ABB RobotStudio station: Celda_4_Enero.rsstn

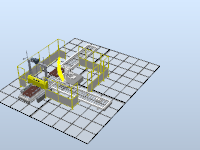
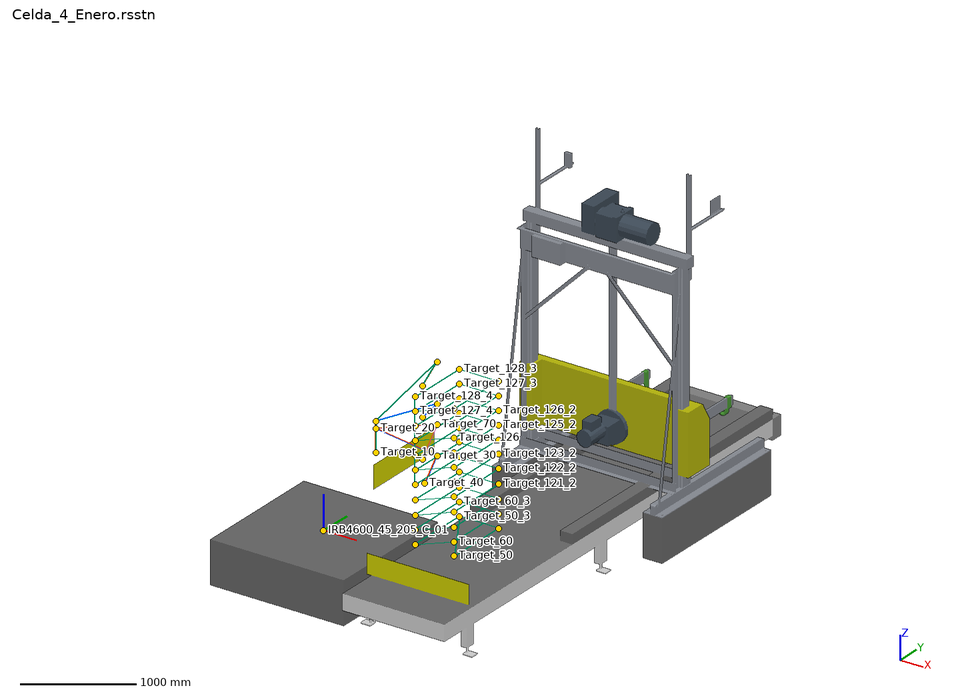
[picture v1: parts stored in the station drawn from their meshes, with robot base, taught points and paths (robot models come from the ABB library and are not in the file)]
Station Celda (saved by RobotStudio 21.3.9648.0)
Controller Controlador1, task T_ROB1: task frame (RAPID world) sits at (0, 0, 435) mm in the station
Controller Controlador1
  mechanical unit ROB_1: IRB4600_45_205_C_01, 6 joints, base frame (0, 0, 0) mm
Layout (positions relative to the parent item):
  - Entrada de canastillas [smart component]
      signals: DO Canasta_ok, DI Soltar, DI Agarrar, DO Agarrado, DI Pallet_fisica
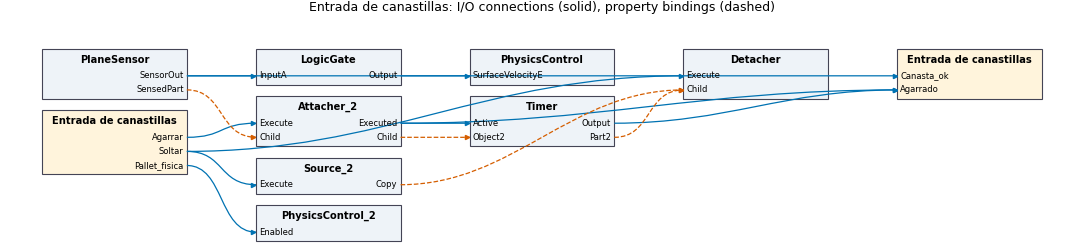
      connections:
        PlaneSensor.SensorOut -> LogicGate.InputA
        LogicGate.Output -> PhysicsControl.SurfaceVelocityEnabled
        PlaneSensor.SensorOut -> Entrada de canastillas.Canasta_ok
        Entrada de canastillas.Agarrar -> Attacher_2.Execute
        Attacher_2.Executed -> Timer.Active
        Timer.Output -> Entrada de canastillas.Agarrado
        Attacher_2.Executed -> Entrada de canastillas.Agarrado
        Entrada de canastillas.Soltar -> Detacher.Execute
        Entrada de canastillas.Pallet_fisica -> PhysicsControl_2.Enabled
        Entrada de canastillas.Soltar -> Source_2.Execute
        PlaneSensor.SensedPart => Attacher_2.Child
        CollisionSensor.Part2 => Detacher.Child
        Attacher_2.Child => CollisionSensor.Object2
        Source_2.Copy => Detacher.Child
    - Source_2 [smart component, from Components\Source.rslib]
        properties: Source=Plastic crate; Copy=(none); Parent=(none); Position=[-2.8 1.3 0.565]; Orientation=[3.14159265358979 0 0]; Transient=false; PhysicsBehavior=3
    - PlaneSensor [smart component, from Components\PlaneSensor.rslib]
        properties: Origin=[-0.076705 1.76 0.467165]; Axis1=[0 -0.91 0]; Axis2=[-5E-06 0 0.232835]; SensedPart=(none)
      - _sensorPart_ [part], size 0 x 910 x 232.8 mm
    - PhysicsControl [smart component, from Components\PhysicsControl.rslib]
        properties: Object=Banda_Canastas; Behavior=2; SurfaceVelocity=0.7
    - LogicGate [smart component, from Components\LogicGate.rslib]
        properties: Operator=NOT; Delay=0
    - Attacher_2 [smart component, from Components\Attacher.rslib]
        properties: Parent=MyNewTool; Flange=0; Child=(none); Mount=false; Offset=[0 0 0]; Orientation=[0 0 0]
    - Detacher [smart component, from Components\Detacher.rslib]
        properties: Child=(none); KeepPosition=true
    - PhysicsControl_2 [smart component, from Components\PhysicsControl.rslib]
        properties: Object=Euro Pallet; Behavior=3; SurfaceVelocity=0
  - IRB4600_45_205_C_01 [mechanism, from Robots\IRB4600_45_205_C_G_01.rslib] at (0, 0, 435) mm; joint values [1.8433, 0.6847, 0.3992, 0, 0.4869, -1.2983] (rad or m)
  - MyNewTool [mechanism] at (-362.82, 1298.26, 725.56) mm, rotated rx -180 ry 0 rz 0 deg
      TCP Gripper at (0, 0, 166) mm
      links: NewGripper
  - Perimetro [graphiccomponentgroup]
    - Fence_2503 [graphiccomponentgroup, from Equipment\Fence_2500.rslib] at (3000, 238.8, 0) mm
      - Body 1 [part, from Equipment\Fence_2500.rslib]
      - Body 2 [part, from Equipment\Fence_2500.rslib]
    - Fence_2502 [graphiccomponentgroup, from Equipment\Fence_2500.rslib] at (3000, -2235.69, 0) mm
      - Body 1 [part, from Equipment\Fence_2500.rslib]
      - Body 2 [part, from Equipment\Fence_2500.rslib]
    - Fence_2500 [graphiccomponentgroup, from Equipment\Fence_2500.rslib] at (-2079.28, 2740, 0) mm, rotated rx 0 ry 0 rz -90 deg
      - Body 1 [part, from Equipment\Fence_2500.rslib]
      - Body 2 [part, from Equipment\Fence_2500.rslib]
    - Fence_740_12 [graphiccomponentgroup, from Equipment\Fence_740.rslib] at (3000, -2297.98, 0) mm, rotated rx 0 ry 0 rz 90 deg
      - Body 1 [part, from Equipment\Fence_740.rslib]
      - Body 2 [part, from Equipment\Fence_740.rslib]
    - Fence_740_11 [graphiccomponentgroup, from Equipment\Fence_740.rslib] at (-2100, -2267.47, 0) mm
      - Body 1 [part, from Equipment\Fence_740.rslib]
      - Body 2 [part, from Equipment\Fence_740.rslib]
    - Fence_740_10 [graphiccomponentgroup, from Equipment\Fence_740.rslib] at (82.68, -2200, 0) mm, rotated rx 0 ry 0 rz -90 deg
      - Body 1 [part, from Equipment\Fence_740.rslib]
      - Body 2 [part, from Equipment\Fence_740.rslib]
    - Fence_740_9 [graphiccomponentgroup, from Equipment\Fence_740.rslib] at (-657.15, -2200, 0) mm, rotated rx 0 ry 0 rz -90 deg
      - Body 1 [part, from Equipment\Fence_740.rslib]
      - Body 2 [part, from Equipment\Fence_740.rslib]
    - Fence_740_8 [graphiccomponentgroup, from Equipment\Fence_740.rslib] at (-1386.41, -2200, 0) mm, rotated rx 0 ry 0 rz -90 deg
      - Body 1 [part, from Equipment\Fence_740.rslib]
      - Body 2 [part, from Equipment\Fence_740.rslib]
    - Fence_740_4 [graphiccomponentgroup, from Equipment\Fence_740.rslib] at (-2153.49, -2200, 0) mm, rotated rx 0 ry 0 rz -90 deg
      - Body 1 [part, from Equipment\Fence_740.rslib]
      - Body 2 [part, from Equipment\Fence_740.rslib]
    - Fence_740_3 [graphiccomponentgroup, from Equipment\Fence_740.rslib] at (-2100, -1490.03, 0) mm
      - Body 1 [part, from Equipment\Fence_740.rslib]
      - Body 2 [part, from Equipment\Fence_740.rslib]
    - Fence_740_2 [graphiccomponentgroup, from Equipment\Fence_740.rslib] at (3000, 2740, 0) mm, rotated rx 0 ry 0 rz 90 deg
      - Body 1 [part, from Equipment\Fence_740.rslib]
      - Body 2 [part, from Equipment\Fence_740.rslib]
    - Fence_740 [graphiccomponentgroup, from Equipment\Fence_740.rslib] at (-2100, 2000, 0) mm
      - Body 1 [part, from Equipment\Fence_740.rslib]
      - Body 2 [part, from Equipment\Fence_740.rslib]
    - Gate [graphiccomponentgroup, from Equipment\Fence_Gate.rslib] at (-2100, 728.56, 0) mm, rotated rx 0 ry 0 rz 180 deg
      - Body 1 [part, from Equipment\Fence_Gate.rslib]
      - Body 2 [part, from Equipment\Fence_Gate.rslib]
      - Body 3 [part, from Equipment\Fence_Gate.rslib]
    - Part_2 [part] at (-700, -700, 0) mm, size 1400 x 1400 x 435 mm
    - Soporte1 [part], size 200 x 1630 x 430 mm
    - Soporte2 [part], size 200 x 1630 x 430 mm
  - Plastic crate [part] at (-3299.78, 1300.28, 558.99) mm, rotated rx 179.83 ry 0.16 rz 0.13 deg, size 603.9 x 403.9 x 145.1 mm
  - Entrada de pallets [smart component]
      connections:
        PlaneSensor.SensorOut -> Source.Execute
        PlaneSensor.SensorOut -> LogicGate.InputA
        LogicGate.Output -> PhysicsControl.SurfaceVelocityEnabled
    - Source [smart component, from Components\Source.rslib]
        properties: Source=Euro Pallet; Copy=Euro Pallet_84; Parent=(none); Position=[1.75 2.6 0.44]; Orientation=[0 0 1.5707963267949]; Transient=false; PhysicsBehavior=3
    - PlaneSensor [smart component, from Components\PlaneSensor.rslib]
        properties: Origin=[0.84 -0.55 0.475]; Axis1=[1.07 0 0]; Axis2=[0 0 0.2]; SensedPart=Body 1
      - _sensorPart_ [part], size 1070 x 0 x 200 mm
    - PhysicsControl [smart component, from Components\PhysicsControl.rslib]
        properties: Object=Banda_P_Entrada_S; Behavior=1; SurfaceVelocity=0.5
    - LogicGate [smart component, from Components\LogicGate.rslib]
        properties: Operator=NOT; Delay=0
  - Bandas [graphiccomponentgroup]
    - Banda_Canastas [part, from Equipment\Conveyor 950 4800 h2.rslib] at (-4200, 850, 0) mm
    - Banda_P_Entrada [part] at (900, 4000, 0) mm, rotated rx 0 ry 0 rz -90 deg, size 5049.9 x 1178.5 x 441.9 mm
    - Banda_P_Entrada_S [part], size 1070 x 4920 x 1 mm
    - Banda_P_Salida [part, from Equipment\Conveyor 950 4000 h2.rslib] at (900, -1050, 0) mm, rotated rx 0 ry 0 rz -90 deg
    - Barrera1 [part], size 130 x 3000 x 100 mm
    - Barrera2 [part] at (-2, 0, 0) mm, size 123 x 3000 x 100 mm
  - Euro Pallet [graphiccomponentgroup, from Equipment\Euro Pallet.rslib] at (1762.72, -569.55, 439.14) mm, rotated rx 0 ry 0 rz 89.52 deg
    - Body 1 [part, from Equipment\Euro Pallet.rslib]
  - Euro Pallet_2 [graphiccomponentgroup, from Equipment\Euro Pallet.rslib] at (1757, -550, 440) mm, rotated rx 0 ry 0 rz 90 deg
    - Body 1 [part, from Equipment\Euro Pallet.rslib]
  - DispenserPallet [part] at (1350, 3500, 430) mm, rotated rx 90 ry 0 rz 180 deg, size 1784 x 3045 x 1697.6 mm
  - Euro Pallet_84 [graphiccomponentgroup, from Equipment\Euro Pallet.rslib] at (1773.49, 2601.34, 439.14) mm, rotated rx 0 ry 0 rz 90.55 deg
    - Body 1 [part, from Equipment\Euro Pallet.rslib]
Attachment: MyNewTool is attached to IRB4600_45_205_C_01 / Link6
Attachment: PhysicsControl is attached to Banda_Canastas
Station signals: DO Canasta_ok
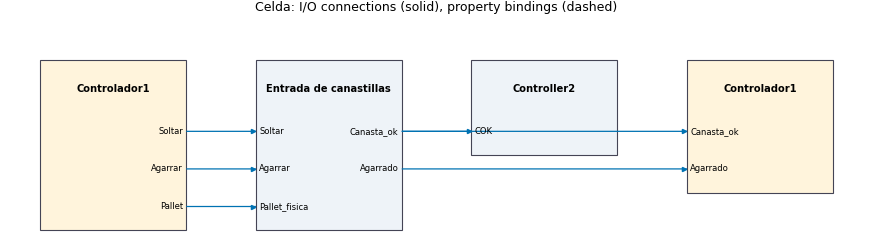
Station logic (signal -> signal, property => property):
  Entrada de canastillas.Canasta_ok -> Controller2.COK
  Entrada de canastillas.Canasta_ok -> Controlador1.Canasta_ok
  Controlador1.Soltar -> Entrada de canastillas.Soltar
  Controlador1.Agarrar -> Entrada de canastillas.Agarrar
  Entrada de canastillas.Agarrado -> Controlador1.Agarrado
  Controlador1.Pallet -> Entrada de canastillas.Pallet_fisica
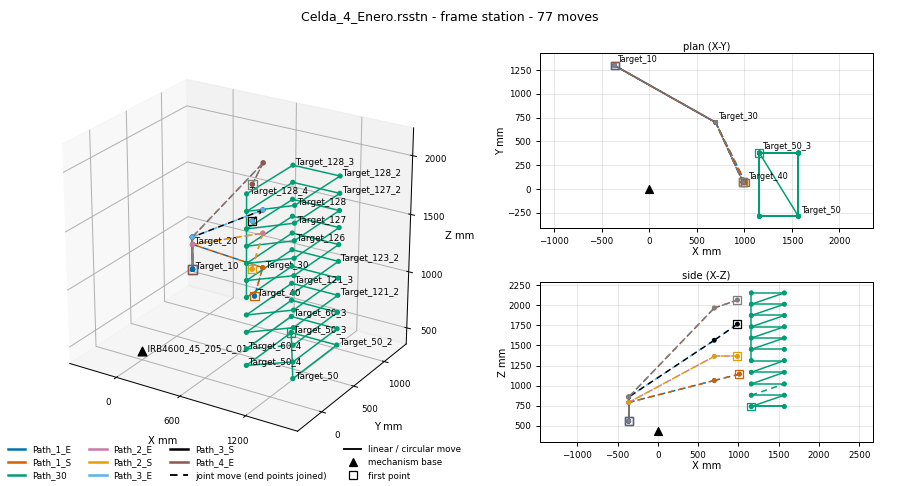
[picture p0: tool path of Celda_4_Enero.rsstn in frame station, 77 of 77 moves have a stored position in this frame; points joined in program order, loops and branches not executed]
Targets, tools, work objects and paths stored in the station, written as RAPID:
! task (no controller)
MODULE CalibData
  TASK PERS wobjdata Workobject_1:=[FALSE,TRUE,"",[[0,0,0],[1,0,0,0]],[[0,0,0],[1,0,0,0]]];
ENDMODULE

! task T_ROB1
MODULE CalibData
  PERS tooldata Gripper:=[TRUE,[[0,0,166],[1,0,0,0]],[27.5,[0,0,86.1],[1,0,0,0],0.589498,1.412,1.775]];
  TASK PERS wobjdata Workobject_1:=[FALSE,TRUE,"",[[0,0,0],[1,0,0,0]],[[0,0,0],[1,0,0,0]]];
ENDMODULE

! task T_ROB1
MODULE Module1
  CONST robtarget Target_10:=[[-362.824,1298.255,124.558],[0,1,0,0],[0,0,0,0],[9E+09,9E+09,9E+09,9E+09,9E+09,9E+09]];
  CONST robtarget Target_30:=[[699.999971128,699.99999496,629.43677315],[0.000000013,0.714564003,0.699570072,0.000000004],[0,-1,-2,0],[9E+09,9E+09,9E+09,9E+09,9E+09,9E+09]];
  CONST robtarget Target_50:=[[1570,-287,307],[0,0.707106781,0.707106781,0],[-1,0,0,0],[9E+09,9E+09,9E+09,9E+09,9E+09,9E+09]];
  CONST robtarget Target_60:=[[1570,-287,447],[0,0.707106781,0.707106781,0],[0,0,0,0],[9E+09,9E+09,9E+09,9E+09,9E+09,9E+09]];
  CONST robtarget Target_50_3:=[[1160,378,307],[0,0.707106781,0.707106781,0],[0,0,0,0],[9E+09,9E+09,9E+09,9E+09,9E+09,9E+09]];
  CONST robtarget Target_50_4:=[[1160,-287,307],[0,0.707106781,0.707106781,0],[-1,0,0,0],[9E+09,9E+09,9E+09,9E+09,9E+09,9E+09]];
  CONST robtarget Target_50_2:=[[1570,378,307],[0,0.707106781,0.707106781,0],[0,0,0,0],[9E+09,9E+09,9E+09,9E+09,9E+09,9E+09]];
  CONST robtarget Target_10_2:=[[-362.824,1298.255,424.558],[-0.000000012,0.998529603,-0.054209154,0.000000007],[1,0,-1,0],[9E+09,9E+09,9E+09,9E+09,9E+09,9E+09]];
  CONST robtarget Target_60_2:=[[1570,378,447],[0,0.707106781,0.707106781,0],[0,0,1,0],[9E+09,9E+09,9E+09,9E+09,9E+09,9E+09]];
  CONST robtarget Target_60_3:=[[1160,378,447],[0,0.707106781,0.707106781,0],[0,0,1,0],[9E+09,9E+09,9E+09,9E+09,9E+09,9E+09]];
  CONST robtarget Target_60_4:=[[1160,-287,447],[0,0.707106781,0.707106781,0],[-1,0,0,0],[9E+09,9E+09,9E+09,9E+09,9E+09,9E+09]];
  CONST robtarget Target_120_2:=[[1570,378,587],[0,0.707106781,0.707106781,0],[0,0,1,0],[9E+09,9E+09,9E+09,9E+09,9E+09,9E+09]];
  CONST robtarget Target_120_3:=[[1160,378,587],[0,0.707106781,0.707106781,0],[0,0,1,0],[9E+09,9E+09,9E+09,9E+09,9E+09,9E+09]];
  CONST robtarget Target_120_4:=[[1160,-287,587],[0,0.707106781,0.707106781,0],[-1,0,0,0],[9E+09,9E+09,9E+09,9E+09,9E+09,9E+09]];
  CONST robtarget Target_121:=[[1570,-287,732],[0,0.707106781,0.707106781,0],[-1,0,0,0],[9E+09,9E+09,9E+09,9E+09,9E+09,9E+09]];
  CONST robtarget Target_121_2:=[[1570,378,732],[0,0.707106781,0.707106781,0],[0,0,1,0],[9E+09,9E+09,9E+09,9E+09,9E+09,9E+09]];
  CONST robtarget Target_121_3:=[[1160,378,732],[0,0.707106781,0.707106781,0],[0,0,1,0],[9E+09,9E+09,9E+09,9E+09,9E+09,9E+09]];
  CONST robtarget Target_121_4:=[[1160,-287,732],[0,0.707106781,0.707106781,0],[-1,0,0,0],[9E+09,9E+09,9E+09,9E+09,9E+09,9E+09]];
  CONST robtarget Target_122:=[[1570,-287,877],[0,0.707106781,0.707106781,0],[-1,0,0,0],[9E+09,9E+09,9E+09,9E+09,9E+09,9E+09]];
  CONST robtarget Target_122_2:=[[1570,378,877],[0,0.707106781,0.707106781,0],[0,0,1,0],[9E+09,9E+09,9E+09,9E+09,9E+09,9E+09]];
  CONST robtarget Target_122_3:=[[1160,378,877],[0,0.707106781,0.707106781,0],[0,0,1,0],[9E+09,9E+09,9E+09,9E+09,9E+09,9E+09]];
  CONST robtarget Target_122_4:=[[1160,-287,877],[0,0.707106781,0.707106781,0],[-1,0,0,0],[9E+09,9E+09,9E+09,9E+09,9E+09,9E+09]];
  CONST robtarget Target_70_2:=[[699.999994937,700.000110159,929.436793547],[-0.000000013,0.714564003,0.699570072,0.000000004],[0,-1,-2,0],[9E+09,9E+09,9E+09,9E+09,9E+09,9E+09]];
  CONST robtarget Target_123:=[[1570,-287,1017],[0,0.707106781,0.707106781,0],[-1,0,0,0],[9E+09,9E+09,9E+09,9E+09,9E+09,9E+09]];
  CONST robtarget Target_124:=[[1570,-287,1157],[0,0.707106781,0.707106781,0],[-1,0,0,0],[9E+09,9E+09,9E+09,9E+09,9E+09,9E+09]];
  CONST robtarget Target_125:=[[1570,-287,1297],[0,0.707106781,0.707106781,0],[-1,0,0,0],[9E+09,9E+09,9E+09,9E+09,9E+09,9E+09]];
  CONST robtarget Target_126:=[[1570,-287,1437],[0,0.707106781,0.707106781,0],[-1,0,0,0],[9E+09,9E+09,9E+09,9E+09,9E+09,9E+09]];
  CONST robtarget Target_127:=[[1570,-287,1577],[0,0.707106781,0.707106781,0],[-1,0,0,0],[9E+09,9E+09,9E+09,9E+09,9E+09,9E+09]];
  CONST robtarget Target_128:=[[1570,-287,1717],[0,0.707106781,0.707106781,0],[-1,0,0,0],[9E+09,9E+09,9E+09,9E+09,9E+09,9E+09]];
  CONST robtarget Target_123_2:=[[1570,378,1017],[0,0.707106781,0.707106781,0],[0,0,1,0],[9E+09,9E+09,9E+09,9E+09,9E+09,9E+09]];
  CONST robtarget Target_124_2:=[[1570,378,1157],[0,0.707106781,0.707106781,0],[0,0,1,0],[9E+09,9E+09,9E+09,9E+09,9E+09,9E+09]];
  CONST robtarget Target_125_2:=[[1570,378,1297],[0,0.707106781,0.707106781,0],[0,0,1,0],[9E+09,9E+09,9E+09,9E+09,9E+09,9E+09]];
  CONST robtarget Target_126_2:=[[1570,378,1437],[0,0.707106781,0.707106781,0],[0,0,1,0],[9E+09,9E+09,9E+09,9E+09,9E+09,9E+09]];
  CONST robtarget Target_127_2:=[[1570,378,1577],[0,0.707106781,0.707106781,0],[0,0,1,0],[9E+09,9E+09,9E+09,9E+09,9E+09,9E+09]];
  CONST robtarget Target_128_2:=[[1570,378,1717],[0,0.707106781,0.707106781,0],[0,0,1,0],[9E+09,9E+09,9E+09,9E+09,9E+09,9E+09]];
  CONST robtarget Target_123_3:=[[1160,378,1017],[0,0.707106781,0.707106781,0],[0,0,1,0],[9E+09,9E+09,9E+09,9E+09,9E+09,9E+09]];
  CONST robtarget Target_124_3:=[[1160,378,1157],[0,0.707106781,0.707106781,0],[0,0,1,0],[9E+09,9E+09,9E+09,9E+09,9E+09,9E+09]];
  CONST robtarget Target_125_3:=[[1160,378,1297],[0,0.707106781,0.707106781,0],[0,0,1,0],[9E+09,9E+09,9E+09,9E+09,9E+09,9E+09]];
  CONST robtarget Target_126_3:=[[1160,378,1437],[0,0.707106781,0.707106781,0],[0,0,1,0],[9E+09,9E+09,9E+09,9E+09,9E+09,9E+09]];
  CONST robtarget Target_127_3:=[[1160,378,1577],[0,0.707106781,0.707106781,0],[0,0,1,0],[9E+09,9E+09,9E+09,9E+09,9E+09,9E+09]];
  CONST robtarget Target_128_3:=[[1160,378,1717],[0,0.707106781,0.707106781,0],[0,0,1,0],[9E+09,9E+09,9E+09,9E+09,9E+09,9E+09]];
  CONST robtarget Target_123_4:=[[1160,-287,1017],[0,0.707106781,0.707106781,0],[-1,0,0,0],[9E+09,9E+09,9E+09,9E+09,9E+09,9E+09]];
  CONST robtarget Target_124_4:=[[1160,-287,1157],[0,0.707106781,0.707106781,0],[-1,0,0,0],[9E+09,9E+09,9E+09,9E+09,9E+09,9E+09]];
  CONST robtarget Target_125_4:=[[1160,-287,1297],[0,0.707106781,0.707106781,0],[-1,0,0,0],[9E+09,9E+09,9E+09,9E+09,9E+09,9E+09]];
  CONST robtarget Target_126_4:=[[1160,-287,1437],[0,0.707106781,0.707106781,0],[-1,0,0,0],[9E+09,9E+09,9E+09,9E+09,9E+09,9E+09]];
  CONST robtarget Target_127_4:=[[1160,-287,1577],[0,0.707106781,0.707106781,0],[-1,0,0,0],[9E+09,9E+09,9E+09,9E+09,9E+09,9E+09]];
  CONST robtarget Target_128_4:=[[1160,-287,1717],[0,0.707106781,0.707106781,0],[-1,2,-2,1],[9E+09,9E+09,9E+09,9E+09,9E+09,9E+09]];
  CONST robtarget Target_10_3:=[[-362.824,1298.255,124.558],[0,1,0,0],[0,0,0,0],[9E+09,9E+09,9E+09,9E+09,9E+09,9E+09]];
  CONST robtarget Target_20_2:=[[123.294942114,850.000075451,439.015995707],[0.000000013,0.714564003,0.699570072,0.000000004],[0,0,1,0],[9E+09,9E+09,9E+09,9E+09,9E+09,9E+09]];
  CONST robtarget Target_10_4:=[[-362.824,1298.255,124.558],[0,1,0,0],[0,0,0,0],[9E+09,9E+09,9E+09,9E+09,9E+09,9E+09]];
  CONST robtarget Target_40:=[[1012.141019914,68.859882763,709.132396194],[0.000000014,0.714564001,0.699570074,0.000000028],[0,0,-3,0],[9E+09,9E+09,9E+09,9E+09,9E+09,9E+09]];
  CONST robtarget Target_20:=[[-361.331074857,1298.255015663,357.504486712],[0.000000006,0.937903782,0.346895511,-0.000000016],[1,0,-2,0],[9E+09,9E+09,9E+09,9E+09,9E+09,9E+09]];
  CONST robtarget Target_70:=[[700.00000486,700.000107801,929.436838226],[0.000000013,0.714563971,0.699570104,-0.000000014],[0,-1,-3,0],[9E+09,9E+09,9E+09,9E+09,9E+09,9E+09]];
  CONST robtarget Target_40_2:=[[987.25590411,72.978878039,929.436817205],[0.00000003,0.714563992,0.699570083,0.000000024],[0,-1,1,0],[9E+09,9E+09,9E+09,9E+09,9E+09,9E+09]];
  CONST robtarget Target_30_2:=[[699.999992444,700.000011939,1129.436971585],[0.000000013,0.714563994,0.699570081,-0.000000007],[0,-1,-3,0],[9E+09,9E+09,9E+09,9E+09,9E+09,9E+09]];
  CONST robtarget Target_40_2_2:=[[987.255899553,72.978877702,1329.437041905],[0.00000002,0.714563994,0.699570081,0.000000013],[0,-1,1,0],[9E+09,9E+09,9E+09,9E+09,9E+09,9E+09]];
  CONST robtarget Target_30_3:=[[699.999994518,700.000014013,1529.436978926],[0.000000013,0.714563998,0.699570077,0.000000012],[0,-1,-3,0],[9E+09,9E+09,9E+09,9E+09,9E+09,9E+09]];
  CONST robtarget Target_40_2_3:=[[987.255908383,72.978882952,1629.436986878],[-0.000000004,0.714563993,0.699570082,0.000000014],[0,0,1,0],[9E+09,9E+09,9E+09,9E+09,9E+09,9E+09]];
  CONST robtarget Target_120:=[[1570.000098335,-287.000000227,586.999987936],[-0.000000001,0.707106765,0.707106797,-0.000000001],[-1,-1,0,0],[9E+09,9E+09,9E+09,9E+09,9E+09,9E+09]];
  PROC Path_1_E()
    MoveL Target_10,v1000,z100,Gripper\WObj:=Workobject_1;
    MoveJ Target_20,v1000,z100,Gripper\WObj:=Workobject_1;
    MoveJ Target_30,v1000,z100,Gripper\WObj:=Workobject_1;
    MoveJ Target_40,v1000,z100,Gripper\WObj:=Workobject_1;
  ENDPROC
  PROC Path_1_S()
    MoveJ Target_40,v1000,z100,Gripper\WObj:=Workobject_1;
    MoveJ Target_30,v800,z100,Gripper\WObj:=Workobject_1;
    MoveJ Target_20,v1000,z100,Gripper\WObj:=Workobject_1;
    MoveJ Target_10,v600,z100,Gripper\WObj:=Workobject_1;
  ENDPROC
  PROC Path_30()
    MoveL Target_50_3,v1000,z100,Gripper\WObj:=Workobject_1;
    MoveL Target_50,v1000,z100,Gripper\WObj:=Workobject_1;
    MoveL Target_50_2,v1000,z100,Gripper\WObj:=Workobject_1;
    MoveL Target_50_3,v1000,z100,Gripper\WObj:=Workobject_1;
    MoveL Target_50_4,v1000,z100,Gripper\WObj:=Workobject_1;
    MoveL Target_60,v1000,z100,Gripper\WObj:=Workobject_1;
    MoveL Target_60_2,v1000,z100,Gripper\WObj:=Workobject_1;
    MoveL Target_60_3,v1000,z100,Gripper\WObj:=Workobject_1;
    MoveL Target_60_4,v1000,z100,Gripper\WObj:=Workobject_1;
    MoveJ Target_120,v1000,z100,Gripper\WObj:=Workobject_1;
    MoveL Target_120_2,v1000,z100,Gripper\WObj:=Workobject_1;
    MoveL Target_120_3,v1000,z100,Gripper\WObj:=Workobject_1;
    MoveL Target_120_4,v1000,z100,Gripper\WObj:=Workobject_1;
    MoveL Target_121,v1000,z100,Gripper\WObj:=Workobject_1;
    MoveL Target_121_2,v1000,z100,Gripper\WObj:=Workobject_1;
    MoveL Target_121_3,v1000,z100,Gripper\WObj:=Workobject_1;
    MoveL Target_121_4,v1000,z100,Gripper\WObj:=Workobject_1;
    MoveL Target_122,v1000,z100,Gripper\WObj:=Workobject_1;
    MoveL Target_122_2,v1000,z100,Gripper\WObj:=Workobject_1;
    MoveL Target_122_3,v1000,z100,Gripper\WObj:=Workobject_1;
    MoveL Target_122_4,v1000,z100,Gripper\WObj:=Workobject_1;
    MoveL Target_128_4,v1000,z100,Gripper\WObj:=Workobject_1;
    MoveL Target_128_3,v1000,z100,Gripper\WObj:=Workobject_1;
    MoveL Target_128_2,v1000,z100,Gripper\WObj:=Workobject_1;
    MoveL Target_128,v1000,z100,Gripper\WObj:=Workobject_1;
    MoveL Target_127_4,v1000,z100,Gripper\WObj:=Workobject_1;
    MoveL Target_127_3,v1000,z100,Gripper\WObj:=Workobject_1;
    MoveL Target_127_2,v1000,z100,Gripper\WObj:=Workobject_1;
    MoveL Target_127,v1000,z100,Gripper\WObj:=Workobject_1;
    MoveL Target_126_4,v1000,z100,Gripper\WObj:=Workobject_1;
    MoveL Target_126_3,v1000,z100,Gripper\WObj:=Workobject_1;
    MoveL Target_126_2,v1000,z100,Gripper\WObj:=Workobject_1;
    MoveL Target_126,v1000,z100,Gripper\WObj:=Workobject_1;
    MoveL Target_125_4,v1000,z100,Gripper\WObj:=Workobject_1;
    MoveL Target_125_3,v1000,z100,Gripper\WObj:=Workobject_1;
    MoveL Target_125_2,v1000,z100,Gripper\WObj:=Workobject_1;
    MoveL Target_125,v1000,z100,Gripper\WObj:=Workobject_1;
    MoveL Target_124_4,v1000,z100,Gripper\WObj:=Workobject_1;
    MoveL Target_124_3,v1000,z100,Gripper\WObj:=Workobject_1;
    MoveL Target_124_2,v1000,z100,Gripper\WObj:=Workobject_1;
    MoveL Target_124,v1000,z100,Gripper\WObj:=Workobject_1;
    MoveL Target_123_4,v1000,z100,Gripper\WObj:=Workobject_1;
    MoveL Target_123_3,v1000,z100,Gripper\WObj:=Workobject_1;
    MoveL Target_123_2,v1000,z100,Gripper\WObj:=Workobject_1;
    MoveL Target_123,v1000,z100,Gripper\WObj:=Workobject_1;
  ENDPROC
  PROC Path_2_E()
    MoveL Target_10,v1000,z100,Gripper\WObj:=Workobject_1;
    MoveJ Target_20,v1000,z100,Gripper\WObj:=Workobject_1;
    MoveJ Target_70,v1000,z100,Gripper\WObj:=Workobject_1;
    MoveJ Target_40_2,v1000,z100,Gripper\WObj:=Workobject_1;
  ENDPROC
  PROC Path_2_S()
    MoveL Target_40_2,v1000,z100,Gripper\WObj:=Workobject_1;
    MoveJ Target_70,v1000,z100,Gripper\WObj:=Workobject_1;
    MoveJ Target_20,v1000,z100,Gripper\WObj:=Workobject_1;
    MoveJ Target_10,v1000,z100,Gripper\WObj:=Workobject_1;
  ENDPROC
  PROC Path_3_E()
    MoveL Target_10,v1000,z100,Gripper\WObj:=Workobject_1;
    MoveL Target_10_2,v1000,z100,Gripper\WObj:=Workobject_1;
    MoveJ Target_30_2,v1000,z100,Gripper\WObj:=Workobject_1;
    MoveJ Target_40_2_2,v1000,z100,Gripper\WObj:=Workobject_1;
  ENDPROC
  PROC Path_3_S()
    MoveL Target_40_2_2,v1000,z100,Gripper\WObj:=Workobject_1;
    MoveJ Target_30_2,v1000,z100,Gripper\WObj:=Workobject_1;
    MoveJ Target_10_2,v1000,z100,Gripper\WObj:=Workobject_1;
    MoveL Target_10,v1000,z100,Gripper\WObj:=Workobject_1;
  ENDPROC
  PROC Path_4_E()
    MoveL Target_10_4,v1000,z100,Gripper\WObj:=Workobject_1;
    MoveL Target_10_2,v1000,z100,Gripper\WObj:=Workobject_1;
    MoveJ Target_30_3,v1000,z100,Gripper\WObj:=Workobject_1;
    MoveJ Target_40_2_3,v1000,z100,Gripper\WObj:=Workobject_1;
  ENDPROC
  PROC Path_4_S()
    MoveL Target_40_2_3,v1000,z100,Gripper\WObj:=Workobject_1;
    MoveJ Target_30_3,v1000,z100,Gripper\WObj:=Workobject_1;
    MoveJ Target_10_2,v1000,z100,Gripper\WObj:=Workobject_1;
    MoveL Target_10_4,v1000,z100,Gripper\WObj:=Workobject_1;
  ENDPROC
ENDMODULE

